// TwinCAT 3 PLC project PlcTc3JsonXmlSampleJsonSaxWriter
// ProgramVersion: 3.1.4021.2
// libraries:
//   Tc2_Standard, * (Beckhoff Automation GmbH)
//   Tc2_System, * (Beckhoff Automation GmbH)
//   Tc3_JsonXml, * (Beckhoff Automation GmbH)
//   Tc3_Module, * (Beckhoff Automation GmbH)
// project tree:
//   DUTs/ E_JsonStates.TcDUT
//   / PlcTask.TcTTO
//   POUs/ MAIN.TcPOU, JsonSaxHandler.TcPOU
// real-time tasks:
//   TASK PlcTask: cycle T#10ms, priority 20, ADS port 350

CONFIGURATION PlcTc3JsonXmlSampleJsonSaxWriter
    RESOURCE PLC ON TwinCAT3
        TASK PlcTask(INTERVAL := T#10ms, PRIORITY := 20);
        PROGRAM MAIN WITH PlcTask : MAIN;
    END_RESOURCE
END_CONFIGURATION

// ---- DUTs/E_JsonStates.TcDUT
{attribute 'qualified_only'}
{attribute 'strict'}
TYPE E_JsonStates :
(
	JSON_STATE_ONSTARTOBJECT1 := 10,
	JSON_STATE_ONKEY_VALUES := 20,
	JSON_STATE_ONSTARTOBJECT2 := 30,
	JSON_STATE_ONKEY_TIMESTAMP := 40,
	JSON_STATE_ONSTRING := 50,
	JSON_STATE_ONKEY_SENSOR1 := 60,
	JSON_STATE_ONLREAL := 70,
	JSON_STATE_ONKEY_SENSOR2 := 80,
	JSON_STATE_ONUDINT := 90,
	JSON_STATE_ONENDOBJECT1 := 100,
	JSON_STATE_ONENDOBJECT2 := 110,
	JSON_STATE_FINISH := 120
);
END_TYPE

// ---- POUs/MAIN.TcPOU
PROGRAM MAIN
VAR
  	(* JSON document *)
	fbJson 			: FB_JsonSaxReader;
	pJsonParse		: JsonSaxHandler;
	sJsonDoc 		: STRING(255) := '{"Values":{"Timestamp":"2017-04-04T12:42:42","Sensor1":42.42,"Sensor2":42}}';	
END_VAR

fbJson.Parse(sJson := sJsonDoc, ipHdl := pJsonParse);

END_PROGRAM

// ---- POUs/JsonSaxHandler.TcPOU
{attribute 'c++_compatible'}
FUNCTION_BLOCK JsonSaxHandler IMPLEMENTS ITcJsonSaxHandler
VAR_INPUT
END_VAR
VAR_OUTPUT
END_VAR
VAR
	(* Values from JSON - written by callback methods *)	  
	sTimestamp 			: STRING(255);
	Sensor1				: LREAL;
	Sensor2				: DINT;
	
	(* State machine variables *)
	eState				: E_JsonStates;
	
	(* Indicators if an expected property has been found in JSON *)
	bStartObjectFound 	: BOOL;
	bEndObjectFound		: BOOL;
	bValuesFound 		: BOOL;
	bTimestampFound 	: BOOL;
	bTimestampValueFound: BOOL;
	bSensor1Found 		: BOOL;
	bSensor1ValueFound	: BOOL;
	bSensor2Found 		: BOOL;
	bSensor2ValueFound	: BOOL;
	
	(* Error indicators *)
	bError				: BOOL;
	sErrorMsg			: STRING(255);
END_VAR

IF bError THEN
	sErrorMsg := 'JSON message does not equal expected format';
END_IF

{attribute 'show'}
{attribute 'c++_compatible'}
{attribute 'minimal_input_size' := '4'}
{attribute 'pack_mode' := '4'}
{warning 'add method implementation'}
METHOD OnBool : HRESULT
VAR_INPUT
	value	: BOOL;
END_VAR
END_METHOD

{attribute 'show'}
{attribute 'c++_compatible'}
{attribute 'minimal_input_size' := '4'}
{attribute 'pack_mode' := '4'}
{warning 'add method implementation'}
METHOD OnDint : HRESULT
VAR_INPUT
	value	: DINT;
END_VAR
Sensor2 := value;
END_METHOD

{attribute 'show'}
{attribute 'c++_compatible'}
{attribute 'minimal_input_size' := '4'}
{attribute 'pack_mode' := '4'}
{warning 'add method implementation'}
METHOD OnEndArray : HRESULT
VAR_INPUT
	elementCount	: UDINT;
END_VAR
END_METHOD

{attribute 'show'}
{attribute 'c++_compatible'}
{attribute 'minimal_input_size' := '4'}
{attribute 'pack_mode' := '4'}
{warning 'add method implementation'}
METHOD OnEndObject : HRESULT
VAR_INPUT
	memberCount	: UDINT;
END_VAR
IF (eState = 100) THEN
	bEndObjectFound := TRUE;
	eState := 110;  
	ELSE
		IF (eState = 110) THEN
			bEndObjectFound := TRUE;
			eState := 120;
		ELSE
			bError := TRUE;  
	  END_IF			
END_IF
END_METHOD

{attribute 'show'}
{attribute 'c++_compatible'}
{attribute 'minimal_input_size' := '4'}
{attribute 'pack_mode' := '4'}
{warning 'add method implementation'}
METHOD OnKey : HRESULT
VAR_IN_OUT CONSTANT
	key	: STRING;
END_VAR
VAR_INPUT
	len	: UDINT;
END_VAR
IF ((eState = 20)AND(key = 'Values')) THEN
	bValuesFound := TRUE;
	eState := 30;
	ELSE
		IF ((eState = 40)AND(key = 'Timestamp')) THEN
		  bTimestampFound := TRUE;
		  eState := 50;
		ELSE
			IF ((eState = 60)AND(key = 'Sensor1')) THEN
				bSensor1Found := TRUE;
				eState := 70;
			ELSE
				IF ((eState = 80)AND(key = 'Sensor2')) THEN
					bSensor2Found := TRUE;
					eState := 90;
				ELSE
					bError := TRUE;
					Onkey := S_FALSE;
				END_IF				  
			END_IF	  
	  	END_IF
END_IF
END_METHOD

{attribute 'show'}
{attribute 'c++_compatible'}
{attribute 'minimal_input_size' := '4'}
{attribute 'pack_mode' := '4'}
{warning 'add method implementation'}
METHOD OnLint : HRESULT
VAR_INPUT
	value	: LINT;
END_VAR
END_METHOD

{attribute 'show'}
{attribute 'c++_compatible'}
{attribute 'minimal_input_size' := '4'}
{attribute 'pack_mode' := '4'}
{warning 'add method implementation'}
METHOD OnLreal : HRESULT
VAR_INPUT
	value	: LREAL;
END_VAR
IF (eState = 70) THEN
	bSensor1ValueFound := TRUE;
	Sensor1 := value;
	eState := 80;
ELSE
	bError := TRUE;
	OnLreal := S_FALSE;
END_IF
END_METHOD

{attribute 'show'}
{attribute 'c++_compatible'}
{attribute 'minimal_input_size' := '4'}
{attribute 'pack_mode' := '4'}
{warning 'add method implementation'}
METHOD OnNull : HRESULT
END_METHOD

{attribute 'show'}
{attribute 'c++_compatible'}
{attribute 'minimal_input_size' := '4'}
{attribute 'pack_mode' := '4'}
{warning 'add method implementation'}
METHOD OnRawNumber : HRESULT
VAR_IN_OUT CONSTANT
	value	: STRING;
END_VAR
VAR_INPUT
	len	: UDINT;
END_VAR
END_METHOD

{attribute 'show'}
{attribute 'c++_compatible'}
{attribute 'minimal_input_size' := '4'}
{attribute 'pack_mode' := '4'}
{warning 'add method implementation'}
METHOD OnStartArray : HRESULT
END_METHOD

{attribute 'show'}
{attribute 'c++_compatible'}
{attribute 'minimal_input_size' := '4'}
{attribute 'pack_mode' := '4'}
{warning 'add method implementation'}
METHOD OnStartObject : HRESULT
IF (eState = 10) THEN
	bStartObjectFound := TRUE;
	eState := 20;  
	ELSE
		IF (eState = 30) THEN
			bStartObjectFound := TRUE;
			eState := 40;
		ELSE
			bError := TRUE;  
	  END_IF			
END_IF
END_METHOD

{attribute 'show'}
{attribute 'c++_compatible'}
{attribute 'minimal_input_size' := '4'}
{attribute 'pack_mode' := '4'}
{warning 'add method implementation'}
METHOD OnString : HRESULT
VAR_IN_OUT CONSTANT
	value	: STRING;
END_VAR
VAR_INPUT
	len	: UDINT;
END_VAR
IF (eState = 50) THEN
	bTimestampValueFound := TRUE;
	sTimestamp := value;
	eState := 60;
ELSE
	bError := TRUE;
	OnString := S_FALSE;
END_IF
END_METHOD

{attribute 'show'}
{attribute 'c++_compatible'}
{attribute 'minimal_input_size' := '4'}
{attribute 'pack_mode' := '4'}
{warning 'add method implementation'}
METHOD OnUdint : HRESULT
VAR_INPUT
	value	: UDINT;
END_VAR
IF (eState = 90) THEN
	bSensor2ValueFound := TRUE;
	Sensor2 := value;
	eState := 100;
ELSE
	bError := TRUE;
	OnUdint := S_FALSE;
END_IF
END_METHOD

{attribute 'show'}
{attribute 'c++_compatible'}
{attribute 'minimal_input_size' := '4'}
{attribute 'pack_mode' := '4'}
{warning 'add method implementation'}
METHOD OnUlint : HRESULT
VAR_INPUT
	value	: ULINT;
END_VAR
END_METHOD

{attribute 'show'}
{attribute 'c++_compatible'}
{attribute 'minimal_input_size' := '4'}
{attribute 'pack_mode' := '4'}
{warning 'add method implementation'}
METHOD TcAddRef : UDINT
END_METHOD

{attribute 'show'}
{attribute 'c++_compatible'}
{attribute 'minimal_input_size' := '4'}
{attribute 'pack_mode' := '4'}
{warning 'add method implementation'}
METHOD TcQueryInterface : HRESULT
VAR_INPUT
	iid	: REFERENCE TO IID;
	pipItf	: POINTER TO PVOID;
END_VAR
END_METHOD

{attribute 'show'}
{attribute 'c++_compatible'}
{attribute 'minimal_input_size' := '4'}
{attribute 'pack_mode' := '4'}
{warning 'add method implementation'}
METHOD TcRelease : UDINT
END_METHOD

END_FUNCTION_BLOCK
